// TIA Portal project "FB CALENDARIO" (V11)

(* hardware
DEVICE "S7300/ET200 station_1"  SIMATIC 300-Station
   slot 0: "Perfil soporte_0"  Rail  6ES7 390-1***0-0AA0
   slot 2: "PLC_1"  CPU 313C-2 DP  6ES7 313-6CF03-0AB0  V2.6
      slot 0: "Interfaz MPI_1"  MPI
      slot 1: "Interfaz DP_1"  DP
      slot 2: "DI16/DO16_1"  DI16/DO16
      slot 4: "Contaje_1"  Counter
*)

// ===== PLC "PLC_1"  CPU 313C-2 DP =====

VAR_GLOBAL   // PLC tag table "Tabla de variables estándar"
   "Tag_1" AT %I0.0 : Bool;
   "Tag_2" AT %MW10 : Int;
   "SG" AT %MW12 : Int;
   "F60" AT %I0.1 : Bool;
   "Tag_3" AT %MW14 : Int;
   "Tag_4" AT %MW16 : Int;
   "Tag_5" AT %MW20 : Int;
   "Tag_6" AT %MW22 : Int;
END_VAR

DATA_BLOCK "CALENDARIO_DB"   // DB1
{ S7_Optimized_Access := 'FALSE' }
VERSION : 0.1
// stored: InstanceOfName CALENDARIO
"CALENDARIO"
BEGIN
END_DATA_BLOCK

FUNCTION_BLOCK "CALENDARIO"   // FB1, LAD
{ S7_Optimized_Access := 'FALSE' }
VERSION : 0.1
   VAR_INPUT
      CARGAR : Bool;
      "SG." : Int;
      "MIN." : Int;
      "HORAS." : Int;
      DIA : Int;
      MES : Int;
      AÑO : Int;
      "TIM 1" : Timer;
      "TIM 2" : Timer;
   END_VAR
   VAR_OUTPUT
      "SG 1" : Int;
      "MIN._1" : Int;
      "HORAS 1" : Int;
      DIA_1 : Int;
      MES_1 : Int;
      AÑO_1 : Int;
   END_VAR
   VAR
      B0 : Bool;
      B1 : Bool;
      B2 : Bool;
      B3 : Bool;
      B4 : Bool;
      B5 : Bool;
      B6 : Bool;
      B7 : Bool;
      F10 : Bool;
      F11 : Bool;
      F12 : Bool;
      F13 : Bool;
      F14 : Bool;
      F15 : Bool;
      F16 : Bool;
      F17 : Bool;
      F20 : Bool;
      F21 : Bool;
      F22 : Bool;
      F23 : Bool;
      F24 : Bool;
      F25 : Bool;
      F26 : Bool;
      F27 : Bool;
      "CSG." : Int;
      "CMIN." : Int;
      CHORAS : Int;
      CDIA : Int;
      CMES : Int;
      CAÑO : Int;
      DRESULTADO : Int;
      MRESULTADO : Int;
      RESULTADO : Int;
   END_VAR
BEGIN
END_FUNCTION_BLOCK

ORGANIZATION_BLOCK "Main"   // OB1, LAD
TITLE = "Main Program Sweep (Cycle)"
{ S7_Optimized_Access := 'FALSE' }
VERSION : 0.1
   VAR_TEMP
      OB1_EV_CLASS : Byte;   // Bits 0-3 = 1 (Coming event), Bits 4-7 = 1 (Event class 1)
      OB1_SCAN_1 : Byte;   // 1 (Cold restart scan 1 of OB 1), 3 (Scan 2-n of OB 1)
      OB1_PRIORITY : Byte;   // Priority of OB Execution
      OB1_OB_NUMBR : Byte;   // 1 (Organization block 1, OB1)
      OB1_RESERVED_1 : Byte;   // Reserved for system
      OB1_RESERVED_2 : Byte;   // Reserved for system
      OB1_PREV_CYCLE : Int;   // Cycle time of previous OB1 scan (milliseconds)
      OB1_MIN_CYCLE : Int;   // Minimum cycle time of OB1 (milliseconds)
      OB1_MAX_CYCLE : Int;   // Maximum cycle time of OB1 (milliseconds)
      OB1_DATE_TIME : Date_And_Time;   // Date and time OB1 started
   END_VAR
BEGIN

REGION Network 1
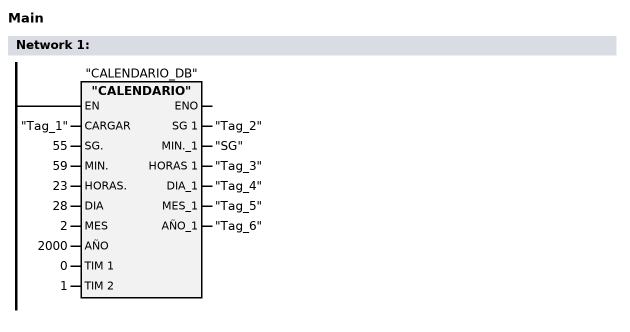
   RUNG wire#powerrail
      "CALENDARIO_DB"(CARGAR := "Tag_1", "SG." := 55, "MIN." := 59, "HORAS." := 23, DIA := 28, MES := 2, AÑO := 2000, "TIM 1" := 0, "TIM 2" := 1, "SG 1" => "Tag_2", "MIN._1" => "SG", "HORAS 1" => "Tag_3", DIA_1 => "Tag_4", MES_1 => "Tag_5", AÑO_1 => "Tag_6")
   END_RUNG
   // the same network as SCL:
   "CALENDARIO_DB"(CARGAR := "Tag_1",   // "CALENDARIO"
                   "SG." := 55,
                   "MIN." := 59,
                   "HORAS." := 23,
                   DIA := 28,
                   MES := 2,
                   AÑO := 2000,
                   "TIM 1" := 0,
                   "TIM 2" := 1,
                   "SG 1" => "Tag_2",
                   "MIN._1" => "SG",
                   "HORAS 1" => "Tag_3",
                   DIA_1 => "Tag_4",
                   MES_1 => "Tag_5",
                   AÑO_1 => "Tag_6");
END_REGION
END_ORGANIZATION_BLOCK